(* PLC project servo_position, Dassault Systèmes ControlBuild 2024x *)
(* stored: creationDateTime 2023-10-04T11:03:54-01:00 *)

(* This module controls positioning behavior of the motion drive *)
FUNCTION_BLOCK motion_control.servo_position
  VAR_INPUT
    MoveAbsEnable : BOOL := false;
    MoveAbsStart : BOOL := false;
    MovePosition : REAL := 0.0;
    MoveSpeed : REAL := 100.0;
    MoveAcceleration : REAL := 100.0;
    MoveDeceleration : REAL := 100.0;
    MAX_SPEED : REAL(0.0..3.4e+38) := 1000.0;
    MAX_ACCEL : REAL(0.0..3.4e+38) := 300.0;
    MAX_DECEL : REAL(0.0..3.4e+38) := 300.0;
    MODULO_LENGTH : REAL := 0.0;
  END_VAR
  VAR_IN_OUT
    status : INT := 0;
    errorFlag : INT := 0;
    MoveAbsDone : BOOL := false;
    ActualPositionAx : REAL := 0.0;
    ActualVelocity : REAL := 0.0;
  END_VAR
  VAR
    firstStep : BOOL := true;
    stepDone : BOOL := false;
  END_VAR
  VAR
    timeToStop : REAL := 0.0;
    distanceToStop : REAL := 0.0;
    distance : REAL := 0.0;
    currentTime : REAL := 0.0;
    currentSpeed1 : REAL := 0.0;
    targetPosition : REAL := 0.0;
  END_VAR
  VAR
    ActualPositionAx1 : REAL := 0.0;
    acceleration : REAL := 0.0;
    deceleration : REAL := 0.0;
    orderSpeed : REAL := 0.0;
    moveDirection : REAL := 0.0;
    moveDirection1 : REAL := 0.0;
    endChangeSpeed : REAL := 0.0;
    ActualVelocity1 : REAL := 0.0;
  END_VAR


ACTION C_source_code:
/* ----------------------------------------------------------------	*/
/* Type : Model of Operative Behaviour					*/
/* Category :  motion control						*/
/* Author : 									*/
/* Update date : June 2021							*/
/* ----------------------------------------------------------------	*/
/* This module controls positioning behavior of the motion drive	*/
/* ----------------------------------------------------------------	*/ 
stepDone = 0;

if (MoveAbsEnable) {
	if (status == 0) {
		stepDone = 1;
		if (MoveAbsStart == 1) {
			errorFlag = 0;
			if (!(MoveAcceleration > 0 && MoveAcceleration <= 100.0)) {
				errorFlag = 1;
			}
			if (!(MoveDeceleration > 0 && MoveDeceleration <= 100.0)) {
				errorFlag = 2;
			}
			if (!(MoveSpeed >= -100.0 && MoveSpeed <= 100.0)) {
				errorFlag = 3;
			}
			if (errorFlag == 0) {
				targetPosition = MovePosition;
				status = 1;
				MoveAbsDone = 0;
				ActualVelocity = 0;
				currentTime = 0;
				acceleration = MoveAcceleration * MAX_ACCEL / 100.0; deceleration = MoveDeceleration * -MAX_DECEL / 100.0; orderSpeed = MoveSpeed * MAX_SPEED / 100.0;
				if (targetPosition == ActualPositionAx) { // test if movement is null
					status = 4;
				} else {
					if (targetPosition < ActualPositionAx) {
						acceleration = -MoveAcceleration * MAX_ACCEL / 100.0; deceleration = -MoveDeceleration * -MAX_DECEL / 100.0; orderSpeed = -MoveSpeed * MAX_SPEED / 100.0;
					}
					endChangeSpeed = orderSpeed  / acceleration;
					// test if movement is very small
					ActualVelocity = ActualVelocity + acceleration * CLOCK_PERIOD/1000000;
					if (orderSpeed > 0 && ActualVelocity > orderSpeed) ActualVelocity = orderSpeed;
					if (orderSpeed < 0 && ActualVelocity < orderSpeed) ActualVelocity = orderSpeed;
					ActualPositionAx = ActualPositionAx + ActualVelocity * CLOCK_PERIOD/1000000;
					distance = (acceleration > 0 ? 1.0 : -1.0) * (targetPosition - ActualPositionAx);
					if ( distance < 0) {
						status = 4;
					}
				}
			}
		}
	}
	
	if (status == 1 && stepDone == 0) { // Acceleration
		stepDone = 1;
		ActualVelocity = ActualVelocity + acceleration * CLOCK_PERIOD/1000000;
		if (orderSpeed > 0 && ActualVelocity > orderSpeed) ActualVelocity = orderSpeed;
		if (orderSpeed < 0 && ActualVelocity < orderSpeed) ActualVelocity = orderSpeed;
		ActualPositionAx = ActualPositionAx + ActualVelocity * CLOCK_PERIOD/1000000;
		timeToStop = fabs(ActualVelocity  / deceleration);
		distanceToStop = (deceleration < 0 ? -1.0 : 1.0) * 0.5 * deceleration * timeToStop * timeToStop;
		distance = (acceleration > 0 ? 1.0 : -1.0) * (targetPosition - ActualPositionAx);
		if (distance <= distanceToStop) {
			status = 3;
		}
		if (currentTime > endChangeSpeed) {
			ActualVelocity = orderSpeed;
			status = 2;
		}
		if (MoveAbsStart == 0 || MoveAbsEnable == 0) {
			status = 6;
		}
	}
	if (status == 2 && stepDone == 0) { // constant speed
		stepDone = 1;
		ActualVelocity = orderSpeed;
		ActualPositionAx = ActualPositionAx + ActualVelocity * CLOCK_PERIOD/1000000;
		timeToStop = fabs(ActualVelocity  / deceleration);
		distanceToStop = (deceleration < 0 ? -1.0 : 1.0) * 0.5 * deceleration * timeToStop * timeToStop;
		distance = (acceleration > 0 ? 1.0 : -1.0) * (targetPosition - ActualPositionAx);
		if (distance <= distanceToStop) {
			status = 3;
		}
		if (MoveAbsStart == 0 || MoveAbsEnable == 0) {
			status = 6;
		}
	}
	if (status == 3 && stepDone == 0) { // deceleration
		stepDone = 1;
		ActualVelocity = ActualVelocity + deceleration * CLOCK_PERIOD/1000000;
		if ((ActualVelocity * deceleration ) >= 0.0) {
			ActualVelocity = currentSpeed1;
		}
		ActualPositionAx = ActualPositionAx + ActualVelocity * CLOCK_PERIOD/1000000;
		timeToStop = fabs(ActualVelocity  / deceleration);
		distanceToStop = (deceleration < 0 ? -1.0 : 1.0) * 0.5 * deceleration * timeToStop * timeToStop;
		distance = (acceleration > 0 ? 1.0 : -1.0) * (targetPosition - ActualPositionAx);
		if ( distance < 0) {
			ActualPositionAx = targetPosition;
			status = 4;
		}
		if (MoveAbsStart == 0 || MoveAbsEnable == 0) {
			status = 6;
		}
	}
	if (status == 4 && stepDone == 0) { // movement succedeed - end OK
		stepDone = 1;
		MoveAbsDone = 1;
		ActualPositionAx = targetPosition;
		ActualVelocity = 0.0;
		status = 5;
	}
	
	if (status == 5 && stepDone == 0) { // terminate protocol handshaking
		stepDone = 1;
		if (MoveAbsStart == 0) {
			MoveAbsDone = 0;
			status = 0;
		}
	}

	if (status == 6 && stepDone == 0) { // movement aborted - deceleration - not reached the position
		stepDone = 1;
		ActualVelocity = ActualVelocity + deceleration * CLOCK_PERIOD/1000000;
		ActualPositionAx = ActualPositionAx + ActualVelocity * CLOCK_PERIOD/1000000;
		if (ActualVelocity1 * ActualVelocity <= 0.0) {
			ActualVelocity = 0;
			status = 0;
		}
	}
}

moveDirection = ActualPositionAx - ActualPositionAx1;

ActualPositionAx1 = ActualPositionAx;
moveDirection1 = moveDirection;
ActualVelocity1 = ActualVelocity;
currentTime += CLOCK_PERIOD/1000000;
currentSpeed1 = ActualVelocity;

firstStep = 0;
END_ACTION
END_FUNCTION_BLOCK
